ADAPTER EVENT_HS_ACK (* Handshake family, request/confirm only (dataless): CNF in, REQ out, no IND/RSP *)
  (* Standard: 61499-1; Description: Copyright (c) 2026 HR Agrartechnik GmbH This program and the accompanying materials are made available under the terms of the Eclipse Public License 2.0 which is available at https://www.eclipse.org/legal/epl-2.0/ SPDX-License-Identifier: EPL-2.0 *)
  (* Version 1.0, 2026-09-02, Franz Höpfinger, HR Agrartechnik GmbH, Reduction of EVENT_HS to just the request/confirm half: REQ/CNF, no IND/RSP - use when the Socket side never needs to send unsolicited indications back to the Plug *)
  PACKAGE adapter::types::bidirectional::Handshake;
  (* Documentation:
  Reduced member of the EVENT_HS family (Handshake design pattern, IEC 61499 primer course, Module 6, Valeriy Vyatkin) that keeps only the request/confirm half of the full REQ/CNF/IND/RSP vocabulary:
    - REQ – request from Plug to Socket ("please do X")
   - CNF – confirmation from Socket to Plug, answers a REQ ("X done")
    No IND/RSP: the Socket side can only ever answer a REQ, it can never push an unsolicited indication back to the Plug. This is a real (if one-directional-per-transaction) handshake, unlike EVENT_HS_UNI - every REQ does get a CNF.
   Same Socket/Plug role split as EVENT_HS: Plug (Name>>) keeps the declared direction and plays the Requester/client role: it fires REQ and reacts to CNF. Socket (>>Name) mirrors the direction and plays the Responder/server role: it reacts to REQ and fires CNF.
   See test_AX/Meins/DesingPatterns/HandshakePattern/HandshakePattern.md for the full write-up of the EVENT_HS family, including this and the other three reduced variants (EVENT_HS_UNI, EVENT_HS_UNI_WSTRING, EVENT_HS_ACK_WSTRING).
  *)
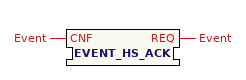
  EVENT_INPUT
    CNF; (* Confirmation from Socket to Plug, answers a REQ *)
  END_EVENT
  EVENT_OUTPUT
    REQ; (* Request from Plug to Socket *)
  END_EVENT
  SERVICE PLUG/SOCKET
    SEQUENCE request_confirm
      PLUG.REQ() -> SOCKET.REQ();
      SOCKET.CNF() -> PLUG.CNF();
    END_SEQUENCE
  END_SERVICE
END_ADAPTER
